TYPE ST_ENCODER_IN :
STRUCT
	bEnable				: BOOL;
END_STRUCT
END_TYPE

(* stored: Version 1.1.0.1
   DUT ST_ENCODER_IN: Id {59649905-68fe-4cff-90be-e0aa91ebcfd4} *)
